FUNCTION CallHardware : BOOL //only purpose of this function is to call modules from Hardware
VAR_STAT
	tempLeft, tempRight : INT;
END_VAR

robot1();	
robot2();

skidA21Left(slots := skidHmiA21Left);
skidA21Right(slots := skidHmiA21Right);

stagingTableLeft(slots := tableHmiA21Left);
stagingTableRight(slots := tableHmiA21Right);

magazineA21Left(slots := magazineHmiA21Left);
magazineA21Right(slots := magazineHmiA21Right);

strapperA21();

verticalDriveA21Left();
horizontalDriveA21Left();

verticalDriveA21Right();
horizontalDriveA21Right();

pistonA21Bottom();

insertionA21Left(
	enable:= TRUE, 
	slider:= verticalDriveA21Left, 
	screw:= horizontalDriveA21Left, 
	softContact=> , 
	active=> , 
	error=> , 
	home=> , 
	homingComplete=> , 
	sliderPos=> );
	
insertionA21Left(
	enable:= TRUE, 
	slider:= verticalDriveA21Right, 
	screw:= horizontalDriveA21Right, 
	softContact=> , 
	active=> , 
	error=> , 
	home=> , 
	homingComplete=> , 
	sliderPos=> );

END_FUNCTION

(* stored: Version 1.1.0.1, ProductVersion 3.1.4024.11
   POU CallHardware: Id {d53bfde7-ef31-4033-a59e-17a8585cdf25}, SpecialFunc None *)
